TYPE U_MOVER_STATE :
UNION
  stState             : ARRAY[1..MAX_MOVER] OF ST_MOVER_STATE;

  byState   AT %I*    : ARRAY[1..MAX_MOVER] OF
                        ARRAY[1..SIZEOF(ST_MOVER_STATE)] OF BYTE;
END_UNION
END_TYPE

(* stored: Version 1.1.0.1
   DUT U_MOVER_STATE: Id {4f6bdbcb-fd67-4f3f-9454-2f432c8514ad} *)
